// TIA Portal V18 export
VAR_GLOBAL   // PLC tag table "Default tag table"
   Pulse1 AT %ID1000 : DInt;
   System_Byte AT %MB1 : Byte;
   FirstScan AT %M1.0 : Bool;
   DiagStatusUpdate AT %M1.1 : Bool;
   AlwaysTRUE AT %M1.2 : Bool;
   AlwaysFALSE AT %M1.3 : Bool;
   Clock_Byte AT %MB0 : Byte;
   Clock_10Hz AT %M0.0 : Bool;
   Clock_5Hz AT %M0.1 : Bool;
   "Clock_2.5Hz" AT %M0.2 : Bool;
   Clock_2Hz AT %M0.3 : Bool;
   "Clock_1.25Hz" AT %M0.4 : Bool;
   Clock_1Hz AT %M0.5 : Bool;
   "Clock_0.625Hz" AT %M0.6 : Bool;
   "Clock_0.5Hz" AT %M0.7 : Bool;
   Flowmeter_pulse AT %I0.0 : Bool;
   Simulate_pulse AT %Q0.4 : Bool;
   Date_time_trigger AT %M98.6 : Bool;
   PREV_Button AT %I1.3 : Bool;
   ENTER_Button AT %I1.4 : Bool;
   NEXT_Button AT %I1.5 : Bool;
   Pendant_START_Button AT %I0.3 : Bool;
   pendant_STOP_Button AT %I0.4 : Bool;
   emergency_mushroom AT %I0.1 : Bool;
   Capacitive_HLS AT %I0.5 : Bool;
   "in Loading" AT %M6.0 : Bool;
   stop_counting_up AT %M6.1 : Bool;
   "NEXT BUTTON FRONT" AT %M6.2 : Bool;
   "PREV BUTTON FRONT" AT %M6.3 : Bool;
   Pendant_emergency_stop AT %I0.2 : Bool;
   FCV_valve_closed AT %I0.6 : Bool;
   ESD_valve_closed AT %I0.7 : Bool;
   ESD_valve_open AT %I1.0 : Bool;
   Ground_monitor_IBC AT %I1.1 : Bool;
   Ground_monitor_truck AT %I1.2 : Bool;
   ESD_solenoid_valve AT %Q0.0 : Bool;
   To_contactor AT %Q0.3 : Bool;
   Flowmeter_analog AT %IW64 : Int;
   spare AT %IW1 : Int;
   "spare 0" AT %Q0.1 : Bool;
   "spare 1" AT %Q0.2 : Bool;
   drained_elapsed_time AT %MW8 : Int;
   RTD_PT100_1 AT %IW0 : Int;
   RTD_PT100_2 AT %IW4 : Int;
   RTD_PT100_3 AT %IW6 : Int;
   stop_counting_down AT %M6.4 : Bool;
END_VAR
